PROGRAM MAIN
VAR
	stDevice1 : ST_Device := (sDeviceName := 'Poco x6', nDeviceValue := 10000);
	stDevice2 : ST_Device := (sDeviceName := 'Samsung s23', nDeviceValue := 30000);
	bToggle : BOOL;
	bNum1 : INT;
END_VAR

END_PROGRAM

(* stored: Version 1.1.0.1, ProductVersion 3.1.4024.16
   POU MAIN: Id {3898c263-ef8a-4860-8627-fa76abac468b}, SpecialFunc None *)
